// This function has been automatically generated from the project information.
{attribute 'signature_flag' := '1073741824'}
{attribute 'TcGenerated'}
{attribute 'no-analysis'}
FUNCTION F_GetCompany : WSTRING
VAR_INPUT
	
END_VAR

F_GetCompany := "RoboConnect";

END_FUNCTION

(* stored: Version 1.1.0.1
   POU F_GetCompany: Id {7f99c8c9-6391-43f7-8b87-5335965ffb92}, SpecialFunc None *)
